SYSTEM VDMA_Station1_Emulator
  (* Version 1.0, 2021-08-05, dorofeev *)
  APPLICATION VDMA_Station1_EmulatorApp
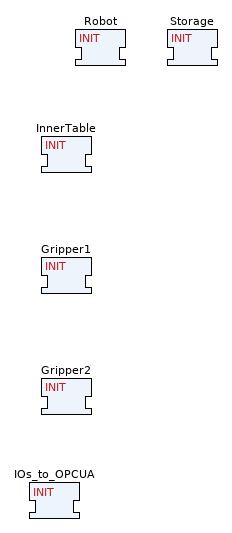
    SUBAPPLICATION Robot
      EVENT_INPUT
        INIT;
      END_EVENT
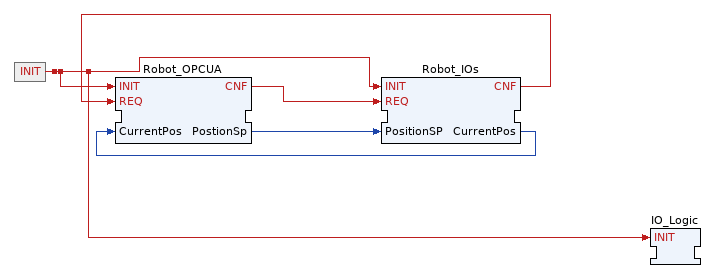
      SUBAPPLICATION IO_Logic
        EVENT_INPUT
          INIT;
        END_EVENT
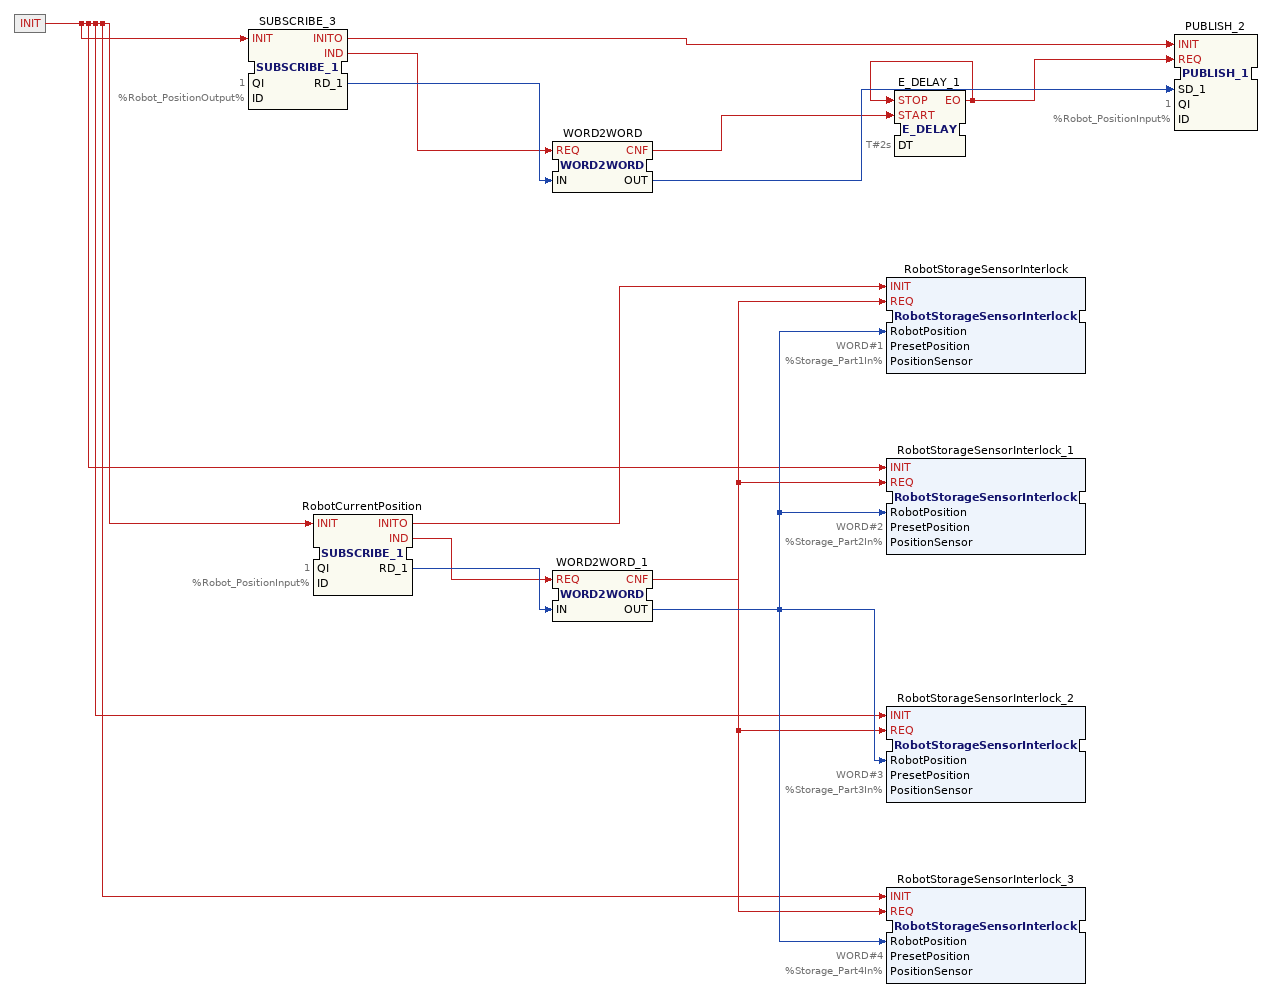
        FBS
          SUBSCRIBE_3 : SUBSCRIBE_1(QI := 1, ID := %Robot_PositionOutput%);
          E_DELAY_1 : E_DELAY(DT := T#2s);
          PUBLISH_2 : PUBLISH_1(QI := 1, ID := %Robot_PositionInput%);
          RobotCurrentPosition : SUBSCRIBE_1(QI := 1, ID := %Robot_PositionInput%);
          WORD2WORD_1 : WORD2WORD;
          WORD2WORD : WORD2WORD;
        END_FBS
        SUBAPPS
          RobotStorageSensorInterlock : RobotStorageSensorInterlock(PresetPosition := WORD#1, PositionSensor := %Storage_Part1In%);
          RobotStorageSensorInterlock_1 : RobotStorageSensorInterlock(PresetPosition := WORD#2, PositionSensor := %Storage_Part2In%);
          RobotStorageSensorInterlock_2 : RobotStorageSensorInterlock(PresetPosition := WORD#3, PositionSensor := %Storage_Part3In%);
          RobotStorageSensorInterlock_3 : RobotStorageSensorInterlock(PresetPosition := WORD#4, PositionSensor := %Storage_Part4In%);
        END_SUBAPPS
        EVENT_CONNECTIONS
          SUBSCRIBE_3.INITO TO PUBLISH_2.INIT;
          E_DELAY_1.EO TO E_DELAY_1.STOP;
          E_DELAY_1.EO TO PUBLISH_2.REQ;
          INIT TO SUBSCRIBE_3.INIT;
          INIT TO RobotStorageSensorInterlock_1.INIT;
          INIT TO RobotStorageSensorInterlock_2.INIT;
          INIT TO RobotStorageSensorInterlock_3.INIT;
          INIT TO RobotCurrentPosition.INIT;
          RobotCurrentPosition.INITO TO RobotStorageSensorInterlock.INIT;
          WORD2WORD_1.CNF TO RobotStorageSensorInterlock.REQ;
          WORD2WORD_1.CNF TO RobotStorageSensorInterlock_3.REQ;
          WORD2WORD_1.CNF TO RobotStorageSensorInterlock_2.REQ;
          WORD2WORD_1.CNF TO RobotStorageSensorInterlock_1.REQ;
          RobotCurrentPosition.IND TO WORD2WORD_1.REQ;
          SUBSCRIBE_3.IND TO WORD2WORD.REQ;
          WORD2WORD.CNF TO E_DELAY_1.START;
        END_CONNECTIONS
        DATA_CONNECTIONS
          WORD2WORD_1.OUT TO RobotStorageSensorInterlock_3.RobotPosition;
          WORD2WORD_1.OUT TO RobotStorageSensorInterlock_2.RobotPosition;
          WORD2WORD_1.OUT TO RobotStorageSensorInterlock_1.RobotPosition;
          WORD2WORD_1.OUT TO RobotStorageSensorInterlock.RobotPosition;
          RobotCurrentPosition.RD_1 TO WORD2WORD_1.IN;
          SUBSCRIBE_3.RD_1 TO WORD2WORD.IN;
          WORD2WORD.OUT TO PUBLISH_2.SD_1;
        END_CONNECTIONS
      END_SUBAPPLICATION
      SUBAPPLICATION Robot_OPCUA
        EVENT_INPUT
          INIT;
          REQ;
        END_EVENT
        EVENT_OUTPUT
          CNF;
        END_EVENT
        VAR_INPUT
          CurrentPos : WORD;
        END_VAR
        VAR_OUTPUT
          PostionSp : WORD;
        END_VAR
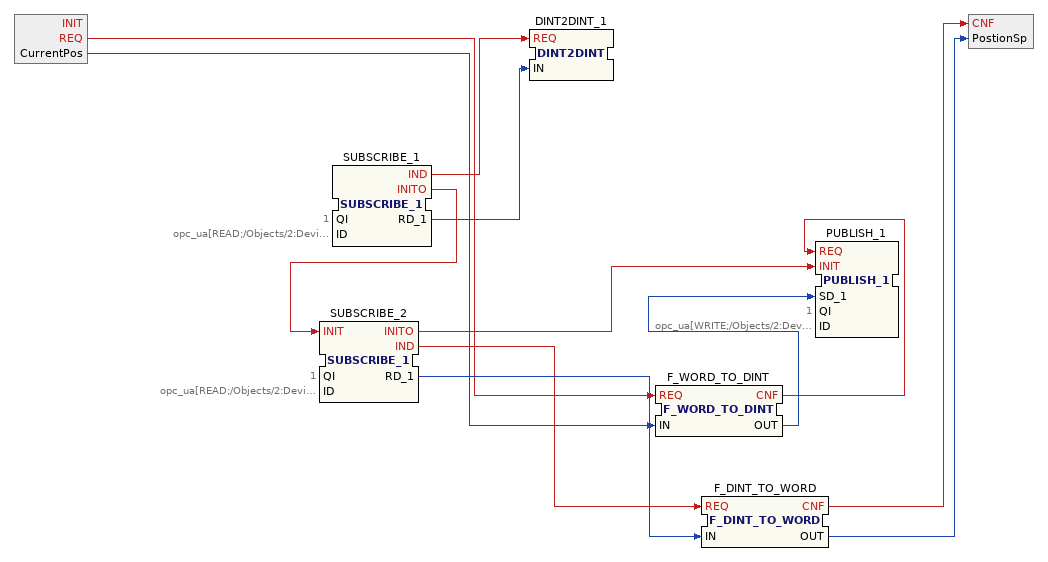
        FBS
          DINT2DINT_1 : DINT2DINT;
          F_WORD_TO_DINT : F_WORD_TO_DINT;
          SUBSCRIBE_2 : SUBSCRIBE_1(QI := 1, ID := opc_ua[READ;/Objects/2:DeviceSet/6:MotionDeviceSystem/5:ProcessData/6:VDMAINVARIABLES/6:SKILL_NMBR]);
          SUBSCRIBE_1 : SUBSCRIBE_1(QI := 1, ID := opc_ua[READ;/Objects/2:DeviceSet/6:MotionDeviceSystem/5:ProcessData/6:VDMAINVARIABLES/6:SKILL_CNTRL]);
          F_DINT_TO_WORD : F_DINT_TO_WORD;
          PUBLISH_1 : PUBLISH_1(QI := 1, ID := opc_ua[WRITE;/Objects/2:DeviceSet/6:MotionDeviceSystem/5:ProcessData/6:VDMAOUTVARIABLES/6:CURRENT_POSITION]);
        END_FBS
        EVENT_CONNECTIONS
          SUBSCRIBE_1.IND TO DINT2DINT_1.REQ;
          F_WORD_TO_DINT.CNF TO PUBLISH_1.REQ;
          SUBSCRIBE_1.INITO TO SUBSCRIBE_2.INIT;
          SUBSCRIBE_2.INITO TO PUBLISH_1.INIT;
          SUBSCRIBE_2.IND TO F_DINT_TO_WORD.REQ;
          REQ TO F_WORD_TO_DINT.REQ;
          F_DINT_TO_WORD.CNF TO CNF;
        END_CONNECTIONS
        DATA_CONNECTIONS
          SUBSCRIBE_1.RD_1 TO DINT2DINT_1.IN;
          F_WORD_TO_DINT.OUT TO PUBLISH_1.SD_1;
          SUBSCRIBE_2.RD_1 TO F_DINT_TO_WORD.IN;
          CurrentPos TO F_WORD_TO_DINT.IN;
          F_DINT_TO_WORD.OUT TO PostionSp;
        END_CONNECTIONS
      END_SUBAPPLICATION
      SUBAPPLICATION Robot_IOs
        EVENT_INPUT
          INIT;
          REQ;
        END_EVENT
        EVENT_OUTPUT
          CNF;
        END_EVENT
        VAR_INPUT
          PositionSP : WORD;
        END_VAR
        VAR_OUTPUT
          CurrentPos : WORD;
        END_VAR
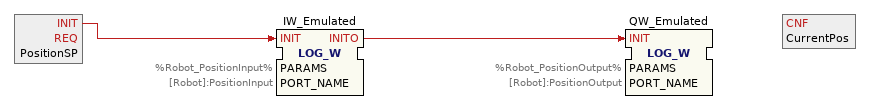
        FBS
          IW_Emulated : LOG_W(PARAMS := %Robot_PositionInput%, PORT_NAME := [Robot]:PositionInput);
          QW_Emulated : LOG_W(PARAMS := %Robot_PositionOutput%, PORT_NAME := [Robot]:PositionOutput);
        END_FBS
        EVENT_CONNECTIONS
          INIT TO IW_Emulated.INIT;
          IW_Emulated.INITO TO QW_Emulated.INIT;
        END_CONNECTIONS
      END_SUBAPPLICATION
      EVENT_CONNECTIONS
        INIT TO Robot_OPCUA.INIT;
        Robot_OPCUA.CNF TO Robot_IOs.REQ;
        INIT TO Robot_IOs.INIT;
        Robot_IOs.CNF TO Robot_OPCUA.REQ;
        INIT TO IO_Logic.INIT;
      END_CONNECTIONS
      DATA_CONNECTIONS
        Robot_OPCUA.PostionSp TO Robot_IOs.PositionSP;
        Robot_IOs.CurrentPos TO Robot_OPCUA.CurrentPos;
      END_CONNECTIONS
    END_SUBAPPLICATION
    SUBAPPLICATION InnerTable
      EVENT_INPUT
        INIT;
      END_EVENT
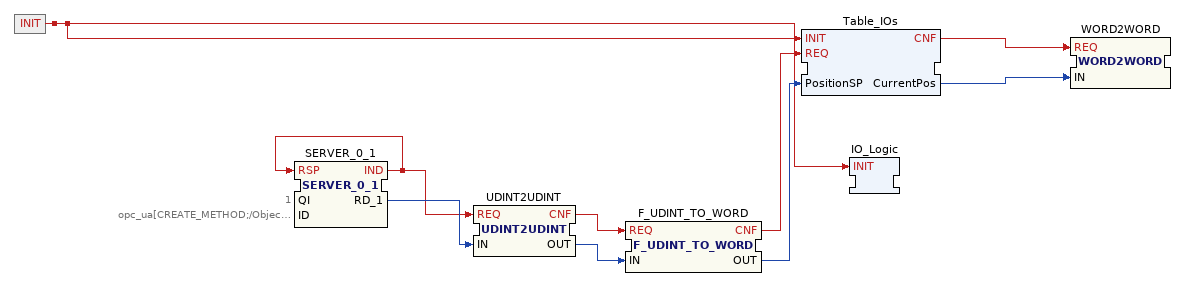
      FBS
        SERVER_0_1 : SERVER_0_1(QI := 1, ID := opc_ua[CREATE_METHOD;/Objects/7:WeissAxis/7:AxisSkillManager/7:MC_MovePresetPosition/7:SetStartParameter]);
        UDINT2UDINT : UDINT2UDINT;
        F_UDINT_TO_WORD : F_UDINT_TO_WORD;
        WORD2WORD : WORD2WORD;
      END_FBS
      SUBAPPLICATION IO_Logic
        EVENT_INPUT
          INIT;
        END_EVENT
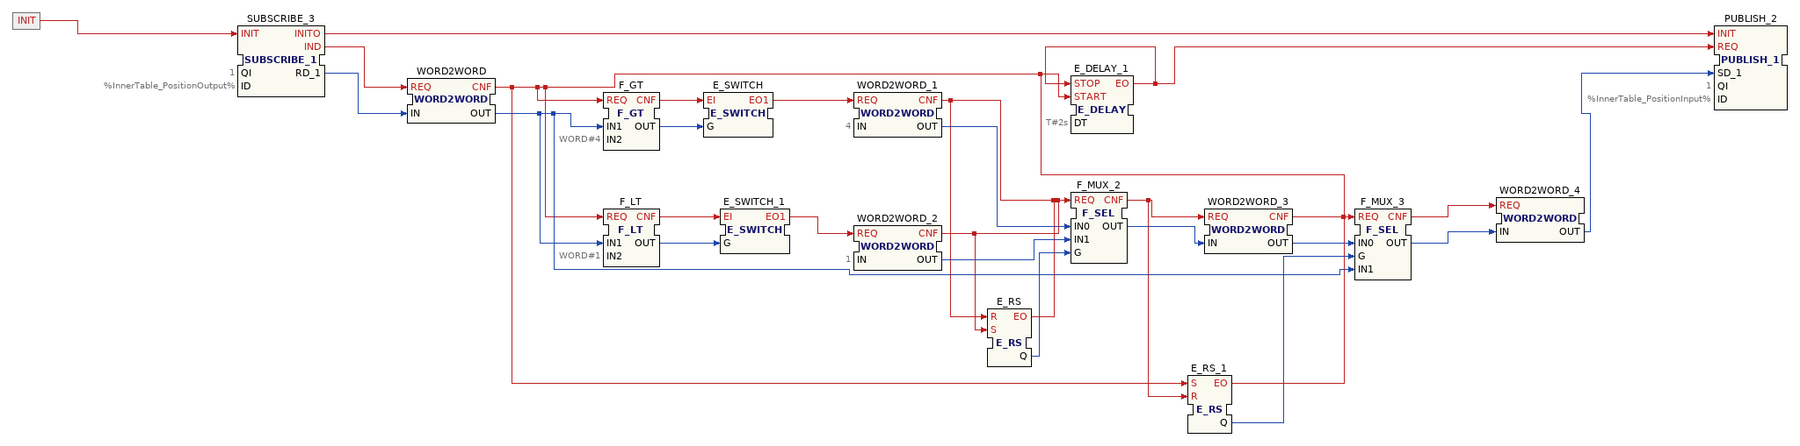
        FBS
          SUBSCRIBE_3 : SUBSCRIBE_1(QI := 1, ID := %InnerTable_PositionOutput%);
          WORD2WORD : WORD2WORD;
          E_DELAY_1 : E_DELAY(DT := T#2s);
          PUBLISH_2 : PUBLISH_1(QI := 1, ID := %InnerTable_PositionInput%);
          F_GT : F_GT(IN2 := WORD#4);
          F_LT : F_LT(IN2 := WORD#1);
          WORD2WORD_1 : WORD2WORD(IN := 4);
          WORD2WORD_2 : WORD2WORD(IN := 1);
          E_SWITCH : E_SWITCH;
          E_SWITCH_1 : E_SWITCH;
          WORD2WORD_3 : WORD2WORD;
          F_MUX_2 : F_SEL;
          F_MUX_3 : F_SEL;
          E_RS : E_RS;
          E_RS_1 : E_RS;
          WORD2WORD_4 : WORD2WORD;
        END_FBS
        EVENT_CONNECTIONS
          SUBSCRIBE_3.INITO TO PUBLISH_2.INIT;
          SUBSCRIBE_3.IND TO WORD2WORD.REQ;
          E_DELAY_1.EO TO E_DELAY_1.STOP;
          E_DELAY_1.EO TO PUBLISH_2.REQ;
          INIT TO SUBSCRIBE_3.INIT;
          WORD2WORD.CNF TO F_GT.REQ;
          WORD2WORD.CNF TO F_LT.REQ;
          F_GT.CNF TO E_SWITCH.EI;
          E_SWITCH.EO1 TO WORD2WORD_1.REQ;
          F_LT.CNF TO E_SWITCH_1.EI;
          E_SWITCH_1.EO1 TO WORD2WORD_2.REQ;
          WORD2WORD.CNF TO E_DELAY_1.START;
          WORD2WORD_1.CNF TO F_MUX_2.REQ;
          WORD2WORD_2.CNF TO F_MUX_2.REQ;
          F_MUX_2.CNF TO WORD2WORD_3.REQ;
          WORD2WORD_3.CNF TO F_MUX_3.REQ;
          WORD2WORD_1.CNF TO E_RS.R;
          WORD2WORD_2.CNF TO E_RS.S;
          E_RS.EO TO F_MUX_2.REQ;
          WORD2WORD.CNF TO E_RS_1.S;
          F_MUX_2.CNF TO E_RS_1.R;
          E_RS_1.EO TO F_MUX_3.REQ;
          F_MUX_3.CNF TO WORD2WORD_4.REQ;
          WORD2WORD.CNF TO F_MUX_3.REQ;
        END_CONNECTIONS
        DATA_CONNECTIONS
          SUBSCRIBE_3.RD_1 TO WORD2WORD.IN;
          WORD2WORD.OUT TO F_LT.IN1;
          WORD2WORD.OUT TO F_GT.IN1;
          F_GT.OUT TO E_SWITCH.G;
          F_LT.OUT TO E_SWITCH_1.G;
          F_MUX_2.OUT TO WORD2WORD_3.IN;
          WORD2WORD_1.OUT TO F_MUX_2.IN0;
          WORD2WORD_2.OUT TO F_MUX_2.IN1;
          WORD2WORD_3.OUT TO F_MUX_3.IN0;
          E_RS.Q TO F_MUX_2.G;
          E_RS_1.Q TO F_MUX_3.G;
          WORD2WORD.OUT TO F_MUX_3.IN1;
          F_MUX_3.OUT TO WORD2WORD_4.IN;
          WORD2WORD_4.OUT TO PUBLISH_2.SD_1;
        END_CONNECTIONS
      END_SUBAPPLICATION
      SUBAPPLICATION Table_IOs
        EVENT_INPUT
          INIT;
          REQ;
        END_EVENT
        EVENT_OUTPUT
          CNF;
        END_EVENT
        VAR_INPUT
          PositionSP : WORD;
        END_VAR
        VAR_OUTPUT
          CurrentPos : WORD;
        END_VAR
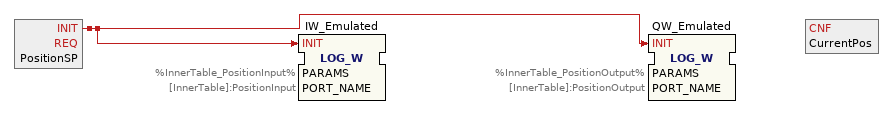
        FBS
          IW_Emulated : LOG_W(PARAMS := %InnerTable_PositionInput%, PORT_NAME := [InnerTable]:PositionInput);
          QW_Emulated : LOG_W(PARAMS := %InnerTable_PositionOutput%, PORT_NAME := [InnerTable]:PositionOutput);
        END_FBS
        EVENT_CONNECTIONS
          INIT TO IW_Emulated.INIT;
          INIT TO QW_Emulated.INIT;
        END_CONNECTIONS
      END_SUBAPPLICATION
      EVENT_CONNECTIONS
        SERVER_0_1.IND TO UDINT2UDINT.REQ;
        INIT TO Table_IOs.INIT;
        INIT TO IO_Logic.INIT;
        UDINT2UDINT.CNF TO F_UDINT_TO_WORD.REQ;
        F_UDINT_TO_WORD.CNF TO Table_IOs.REQ;
        Table_IOs.CNF TO WORD2WORD.REQ;
        SERVER_0_1.IND TO SERVER_0_1.RSP;
      END_CONNECTIONS
      DATA_CONNECTIONS
        SERVER_0_1.RD_1 TO UDINT2UDINT.IN;
        UDINT2UDINT.OUT TO F_UDINT_TO_WORD.IN;
        F_UDINT_TO_WORD.OUT TO Table_IOs.PositionSP;
        Table_IOs.CurrentPos TO WORD2WORD.IN;
      END_CONNECTIONS
    END_SUBAPPLICATION
    SUBAPPLICATION Storage
      EVENT_INPUT
        INIT;
      END_EVENT
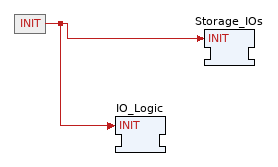
      SUBAPPLICATION IO_Logic
        EVENT_INPUT
          INIT;
        END_EVENT
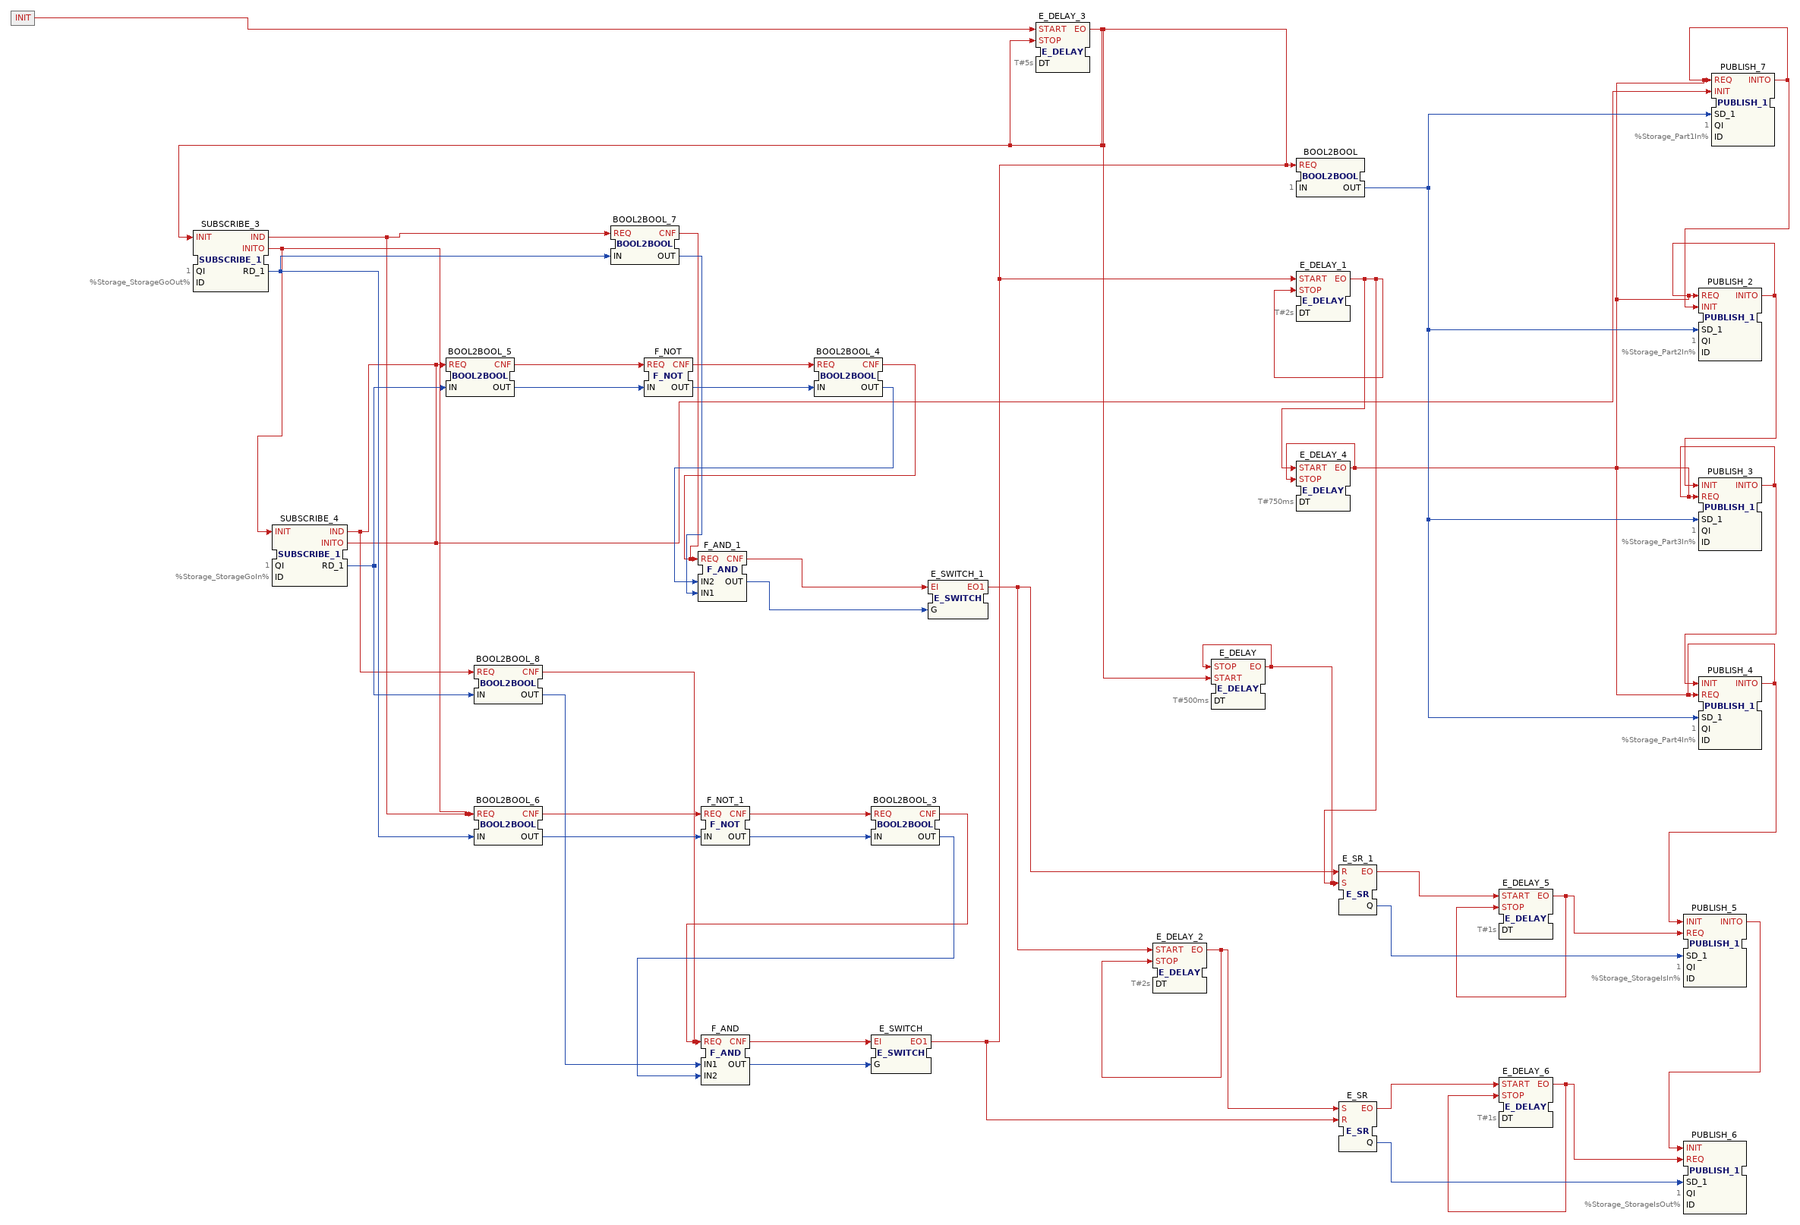
        FBS
          E_SWITCH_1 : E_SWITCH;
          BOOL2BOOL_4 : BOOL2BOOL;
          F_NOT : F_NOT;
          PUBLISH_3 : PUBLISH_1(QI := 1, ID := %Storage_Part3In%);
          BOOL2BOOL_6 : BOOL2BOOL;
          E_SR_1 : E_SR;
          F_NOT_1 : F_NOT;
          PUBLISH_7 : PUBLISH_1(QI := 1, ID := %Storage_Part1In%);
          BOOL2BOOL : BOOL2BOOL(IN := 1);
          BOOL2BOOL_5 : BOOL2BOOL;
          BOOL2BOOL_7 : BOOL2BOOL;
          E_SR : E_SR;
          F_AND_1 : F_AND;
          SUBSCRIBE_4 : SUBSCRIBE_1(QI := 1, ID := %Storage_StorageGoIn%);
          SUBSCRIBE_3 : SUBSCRIBE_1(QI := 1, ID := %Storage_StorageGoOut%);
          PUBLISH_6 : PUBLISH_1(QI := 1, ID := %Storage_StorageIsOut%);
          F_AND : F_AND;
          BOOL2BOOL_3 : BOOL2BOOL;
          PUBLISH_5 : PUBLISH_1(QI := 1, ID := %Storage_StorageIsIn%);
          PUBLISH_4 : PUBLISH_1(QI := 1, ID := %Storage_Part4In%);
          E_DELAY_2 : E_DELAY(DT := T#2s);
          BOOL2BOOL_8 : BOOL2BOOL;
          E_DELAY_1 : E_DELAY(DT := T#2s);
          PUBLISH_2 : PUBLISH_1(QI := 1, ID := %Storage_Part2In%);
          E_SWITCH : E_SWITCH;
          E_DELAY : E_DELAY(DT := T#500ms);
          E_DELAY_3 : E_DELAY(DT := T#5s);
          E_DELAY_4 : E_DELAY(DT := T#750ms);
          E_DELAY_5 : E_DELAY(DT := T#1s);
          E_DELAY_6 : E_DELAY(DT := T#1s);
        END_FBS
        EVENT_CONNECTIONS
          F_AND_1.CNF TO E_SWITCH_1.EI;
          E_SWITCH_1.EO1 TO E_SR_1.R;
          E_SWITCH_1.EO1 TO E_DELAY_2.START;
          F_NOT.CNF TO BOOL2BOOL_4.REQ;
          BOOL2BOOL_4.CNF TO F_AND_1.REQ;
          BOOL2BOOL_5.CNF TO F_NOT.REQ;
          PUBLISH_2.INITO TO PUBLISH_3.INIT;
          PUBLISH_3.INITO TO PUBLISH_3.REQ;
          PUBLISH_3.INITO TO PUBLISH_4.INIT;
          SUBSCRIBE_3.IND TO BOOL2BOOL_6.REQ;
          SUBSCRIBE_3.INITO TO BOOL2BOOL_6.REQ;
          BOOL2BOOL_6.CNF TO F_NOT_1.REQ;
          E_DELAY_1.EO TO E_SR_1.S;
          F_NOT_1.CNF TO BOOL2BOOL_3.REQ;
          PUBLISH_7.INITO TO PUBLISH_7.REQ;
          E_SWITCH.EO1 TO BOOL2BOOL.REQ;
          SUBSCRIBE_4.IND TO BOOL2BOOL_5.REQ;
          SUBSCRIBE_4.INITO TO BOOL2BOOL_5.REQ;
          SUBSCRIBE_3.IND TO BOOL2BOOL_7.REQ;
          BOOL2BOOL_7.CNF TO F_AND_1.REQ;
          E_DELAY_2.EO TO E_SR.S;
          E_SWITCH.EO1 TO E_SR.R;
          SUBSCRIBE_3.INITO TO SUBSCRIBE_4.INIT;
          SUBSCRIBE_4.IND TO BOOL2BOOL_8.REQ;
          PUBLISH_5.INITO TO PUBLISH_6.INIT;
          BOOL2BOOL_3.CNF TO F_AND.REQ;
          BOOL2BOOL_8.CNF TO F_AND.REQ;
          F_AND.CNF TO E_SWITCH.EI;
          PUBLISH_4.INITO TO PUBLISH_5.INIT;
          PUBLISH_4.INITO TO PUBLISH_4.REQ;
          E_DELAY_2.EO TO E_DELAY_2.STOP;
          E_SWITCH.EO1 TO E_DELAY_1.START;
          E_DELAY_1.EO TO E_DELAY_1.STOP;
          PUBLISH_2.INITO TO PUBLISH_2.REQ;
          E_DELAY.EO TO E_DELAY.STOP;
          E_DELAY.EO TO E_SR_1.S;
          E_DELAY_3.EO TO BOOL2BOOL.REQ;
          E_DELAY_3.EO TO E_DELAY.START;
          INIT TO E_DELAY_3.START;
          E_DELAY_3.EO TO E_DELAY_3.STOP;
          E_DELAY_4.EO TO PUBLISH_2.REQ;
          E_DELAY_4.EO TO PUBLISH_4.REQ;
          E_DELAY_4.EO TO PUBLISH_7.REQ;
          E_DELAY_4.EO TO PUBLISH_3.REQ;
          E_DELAY_1.EO TO E_DELAY_4.START;
          E_DELAY_4.EO TO E_DELAY_4.STOP;
          E_SR_1.EO TO E_DELAY_5.START;
          E_DELAY_5.EO TO PUBLISH_5.REQ;
          E_DELAY_5.EO TO E_DELAY_5.STOP;
          E_SR.EO TO E_DELAY_6.START;
          E_DELAY_6.EO TO PUBLISH_6.REQ;
          E_DELAY_6.EO TO E_DELAY_6.STOP;
          E_DELAY_3.EO TO SUBSCRIBE_3.INIT;
          PUBLISH_7.INITO TO PUBLISH_2.INIT;
          SUBSCRIBE_4.INITO TO PUBLISH_7.INIT;
        END_CONNECTIONS
        DATA_CONNECTIONS
          F_AND_1.OUT TO E_SWITCH_1.G;
          F_NOT.OUT TO BOOL2BOOL_4.IN;
          BOOL2BOOL_4.OUT TO F_AND_1.IN2;
          BOOL2BOOL_5.OUT TO F_NOT.IN;
          BOOL2BOOL.OUT TO PUBLISH_3.SD_1;
          SUBSCRIBE_3.RD_1 TO BOOL2BOOL_6.IN;
          BOOL2BOOL_6.OUT TO F_NOT_1.IN;
          F_NOT_1.OUT TO BOOL2BOOL_3.IN;
          BOOL2BOOL.OUT TO PUBLISH_7.SD_1;
          BOOL2BOOL.OUT TO PUBLISH_4.SD_1;
          BOOL2BOOL.OUT TO PUBLISH_2.SD_1;
          SUBSCRIBE_4.RD_1 TO BOOL2BOOL_5.IN;
          SUBSCRIBE_3.RD_1 TO BOOL2BOOL_7.IN;
          BOOL2BOOL_7.OUT TO F_AND_1.IN1;
          E_SR.Q TO PUBLISH_6.SD_1;
          SUBSCRIBE_4.RD_1 TO BOOL2BOOL_8.IN;
          BOOL2BOOL_8.OUT TO F_AND.IN1;
          BOOL2BOOL_3.OUT TO F_AND.IN2;
          F_AND.OUT TO E_SWITCH.G;
          E_SR_1.Q TO PUBLISH_5.SD_1;
        END_CONNECTIONS
      END_SUBAPPLICATION
      SUBAPPLICATION Storage_IOs
        EVENT_INPUT
          INIT;
        END_EVENT
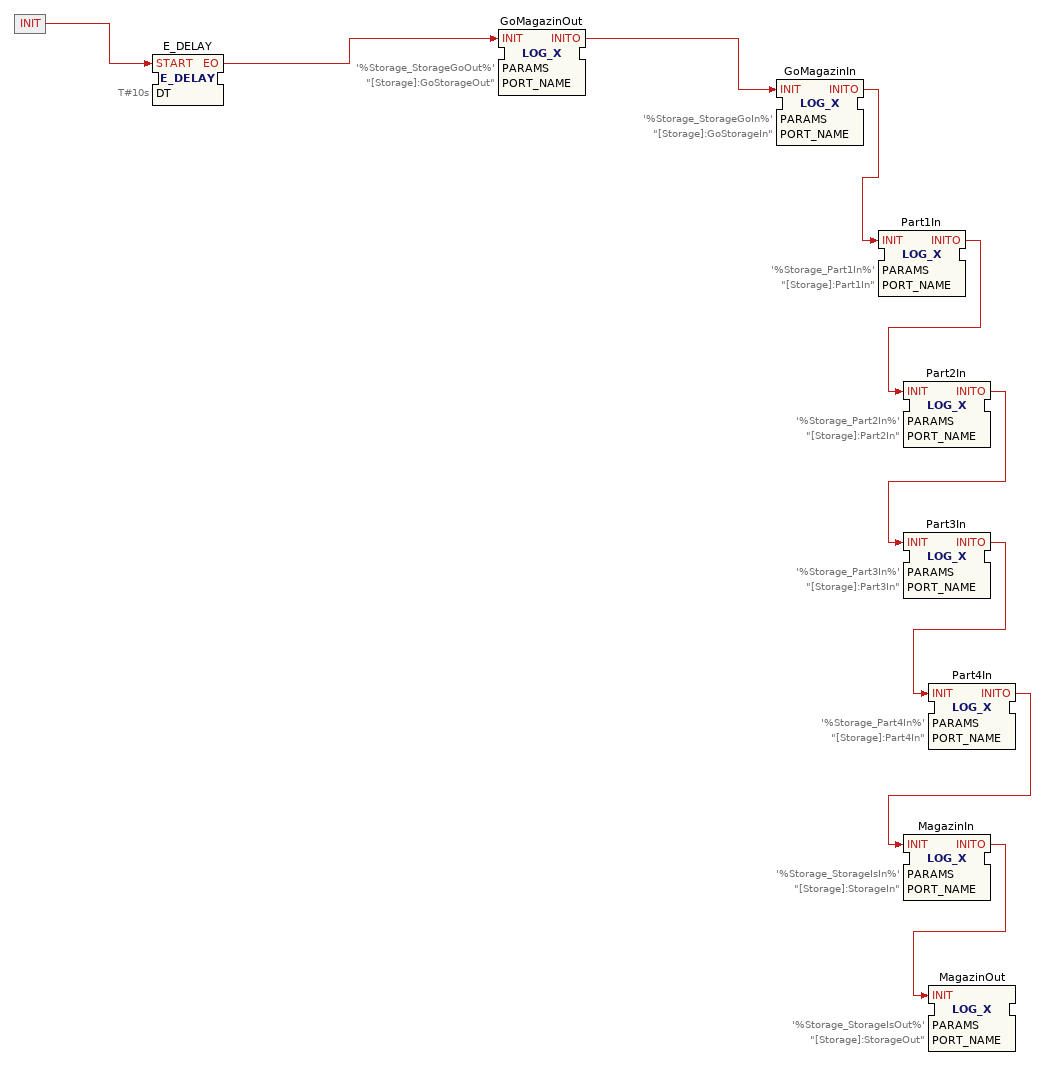
        FBS
          GoMagazinIn : LOG_X(PARAMS := '%Storage_StorageGoIn%', PORT_NAME := "[Storage]:GoStorageIn");
          GoMagazinOut : LOG_X(PARAMS := '%Storage_StorageGoOut%', PORT_NAME := "[Storage]:GoStorageOut");
          Part2In : LOG_X(PARAMS := '%Storage_Part2In%', PORT_NAME := "[Storage]:Part2In");
          Part1In : LOG_X(PARAMS := '%Storage_Part1In%', PORT_NAME := "[Storage]:Part1In");
          Part4In : LOG_X(PARAMS := '%Storage_Part4In%', PORT_NAME := "[Storage]:Part4In");
          Part3In : LOG_X(PARAMS := '%Storage_Part3In%', PORT_NAME := "[Storage]:Part3In");
          MagazinIn : LOG_X(PARAMS := '%Storage_StorageIsIn%', PORT_NAME := "[Storage]:StorageIn");
          MagazinOut : LOG_X(PARAMS := '%Storage_StorageIsOut%', PORT_NAME := "[Storage]:StorageOut");
          E_DELAY : E_DELAY(DT := T#10s);
        END_FBS
        EVENT_CONNECTIONS
          GoMagazinOut.INITO TO GoMagazinIn.INIT;
          GoMagazinIn.INITO TO Part1In.INIT;
          Part1In.INITO TO Part2In.INIT;
          Part2In.INITO TO Part3In.INIT;
          Part3In.INITO TO Part4In.INIT;
          Part4In.INITO TO MagazinIn.INIT;
          MagazinIn.INITO TO MagazinOut.INIT;
          INIT TO E_DELAY.START;
          E_DELAY.EO TO GoMagazinOut.INIT;
        END_CONNECTIONS
      END_SUBAPPLICATION
      EVENT_CONNECTIONS
        INIT TO IO_Logic.INIT;
        INIT TO Storage_IOs.INIT;
      END_CONNECTIONS
    END_SUBAPPLICATION
    SUBAPPLICATION Gripper1
      EVENT_INPUT
        INIT;
      END_EVENT
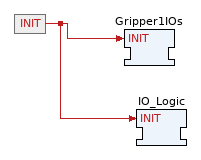
      SUBAPPLICATION Gripper1IOs
        EVENT_INPUT
          INIT;
        END_EVENT
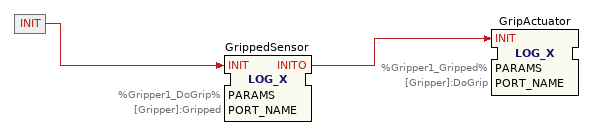
        FBS
          GripActuator : LOG_X(PARAMS := %Gripper1_Gripped%, PORT_NAME := [Gripper]:DoGrip);
          GrippedSensor : LOG_X(PARAMS := %Gripper1_DoGrip%, PORT_NAME := [Gripper]:Gripped);
        END_FBS
        EVENT_CONNECTIONS
          INIT TO GrippedSensor.INIT;
          GrippedSensor.INITO TO GripActuator.INIT;
        END_CONNECTIONS
      END_SUBAPPLICATION
      SUBAPPLICATION IO_Logic
        EVENT_INPUT
          INIT;
        END_EVENT
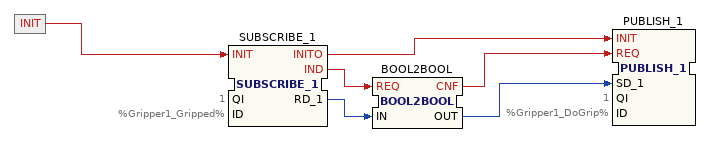
        FBS
          SUBSCRIBE_1 : SUBSCRIBE_1(QI := 1, ID := %Gripper1_Gripped%);
          BOOL2BOOL : BOOL2BOOL;
          PUBLISH_1 : PUBLISH_1(QI := 1, ID := %Gripper1_DoGrip%);
        END_FBS
        EVENT_CONNECTIONS
          SUBSCRIBE_1.INITO TO PUBLISH_1.INIT;
          SUBSCRIBE_1.IND TO BOOL2BOOL.REQ;
          BOOL2BOOL.CNF TO PUBLISH_1.REQ;
          INIT TO SUBSCRIBE_1.INIT;
        END_CONNECTIONS
        DATA_CONNECTIONS
          SUBSCRIBE_1.RD_1 TO BOOL2BOOL.IN;
          BOOL2BOOL.OUT TO PUBLISH_1.SD_1;
        END_CONNECTIONS
      END_SUBAPPLICATION
      EVENT_CONNECTIONS
        INIT TO IO_Logic.INIT;
        INIT TO Gripper1IOs.INIT;
      END_CONNECTIONS
    END_SUBAPPLICATION
    SUBAPPLICATION Gripper2
      EVENT_INPUT
        INIT;
      END_EVENT
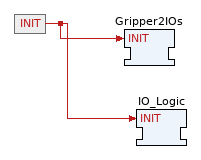
      SUBAPPLICATION Gripper2IOs
        EVENT_INPUT
          INIT;
        END_EVENT
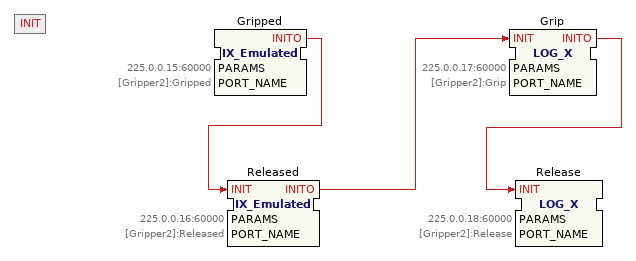
        FBS
          Grip : LOG_X(PARAMS := 225.0.0.17:60000, PORT_NAME := [Gripper2]:Grip);
          Gripped : IX_Emulated(PARAMS := 225.0.0.15:60000, PORT_NAME := [Gripper2]:Gripped);
          Released : IX_Emulated(PARAMS := 225.0.0.16:60000, PORT_NAME := [Gripper2]:Released);
          Release : LOG_X(PARAMS := 225.0.0.18:60000, PORT_NAME := [Gripper2]:Release);
        END_FBS
        EVENT_CONNECTIONS
          Gripped.INITO TO Released.INIT;
          Released.INITO TO Grip.INIT;
          Grip.INITO TO Release.INIT;
        END_CONNECTIONS
      END_SUBAPPLICATION
      SUBAPPLICATION IO_Logic
        EVENT_INPUT
          INIT;
        END_EVENT
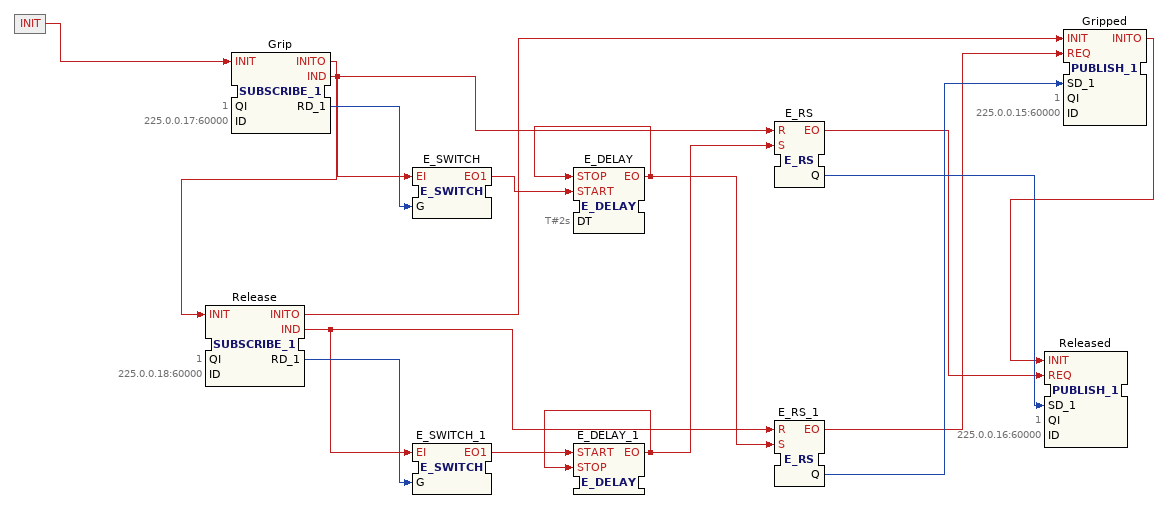
        FBS
          Grip : SUBSCRIBE_1(QI := 1, ID := 225.0.0.17:60000);
          Gripped : PUBLISH_1(QI := 1, ID := 225.0.0.15:60000);
          Release : SUBSCRIBE_1(QI := 1, ID := 225.0.0.18:60000);
          Released : PUBLISH_1(QI := 1, ID := 225.0.0.16:60000);
          E_DELAY : E_DELAY(DT := T#2s);
          E_RS : E_RS;
          E_RS_1 : E_RS;
          E_DELAY_1 : E_DELAY;
          E_SWITCH : E_SWITCH;
          E_SWITCH_1 : E_SWITCH;
        END_FBS
        EVENT_CONNECTIONS
          INIT TO Grip.INIT;
          Grip.INITO TO Release.INIT;
          Release.INITO TO Gripped.INIT;
          Gripped.INITO TO Released.INIT;
          E_DELAY.EO TO E_DELAY.STOP;
          Grip.IND TO E_RS.R;
          E_RS.EO TO Released.REQ;
          Release.IND TO E_RS_1.R;
          E_RS_1.EO TO Gripped.REQ;
          E_DELAY.EO TO E_RS_1.S;
          Grip.IND TO E_SWITCH.EI;
          E_SWITCH.EO1 TO E_DELAY.START;
          Release.IND TO E_SWITCH_1.EI;
          E_SWITCH_1.EO1 TO E_DELAY_1.START;
          E_DELAY_1.EO TO E_DELAY_1.STOP;
          E_DELAY_1.EO TO E_RS.S;
        END_CONNECTIONS
        DATA_CONNECTIONS
          E_RS.Q TO Released.SD_1;
          E_RS_1.Q TO Gripped.SD_1;
          Grip.RD_1 TO E_SWITCH.G;
          Release.RD_1 TO E_SWITCH_1.G;
        END_CONNECTIONS
      END_SUBAPPLICATION
      EVENT_CONNECTIONS
        INIT TO Gripper2IOs.INIT;
        INIT TO IO_Logic.INIT;
      END_CONNECTIONS
    END_SUBAPPLICATION
    SUBAPPLICATION IOs_to_OPCUA
      EVENT_INPUT
        INIT;
      END_EVENT
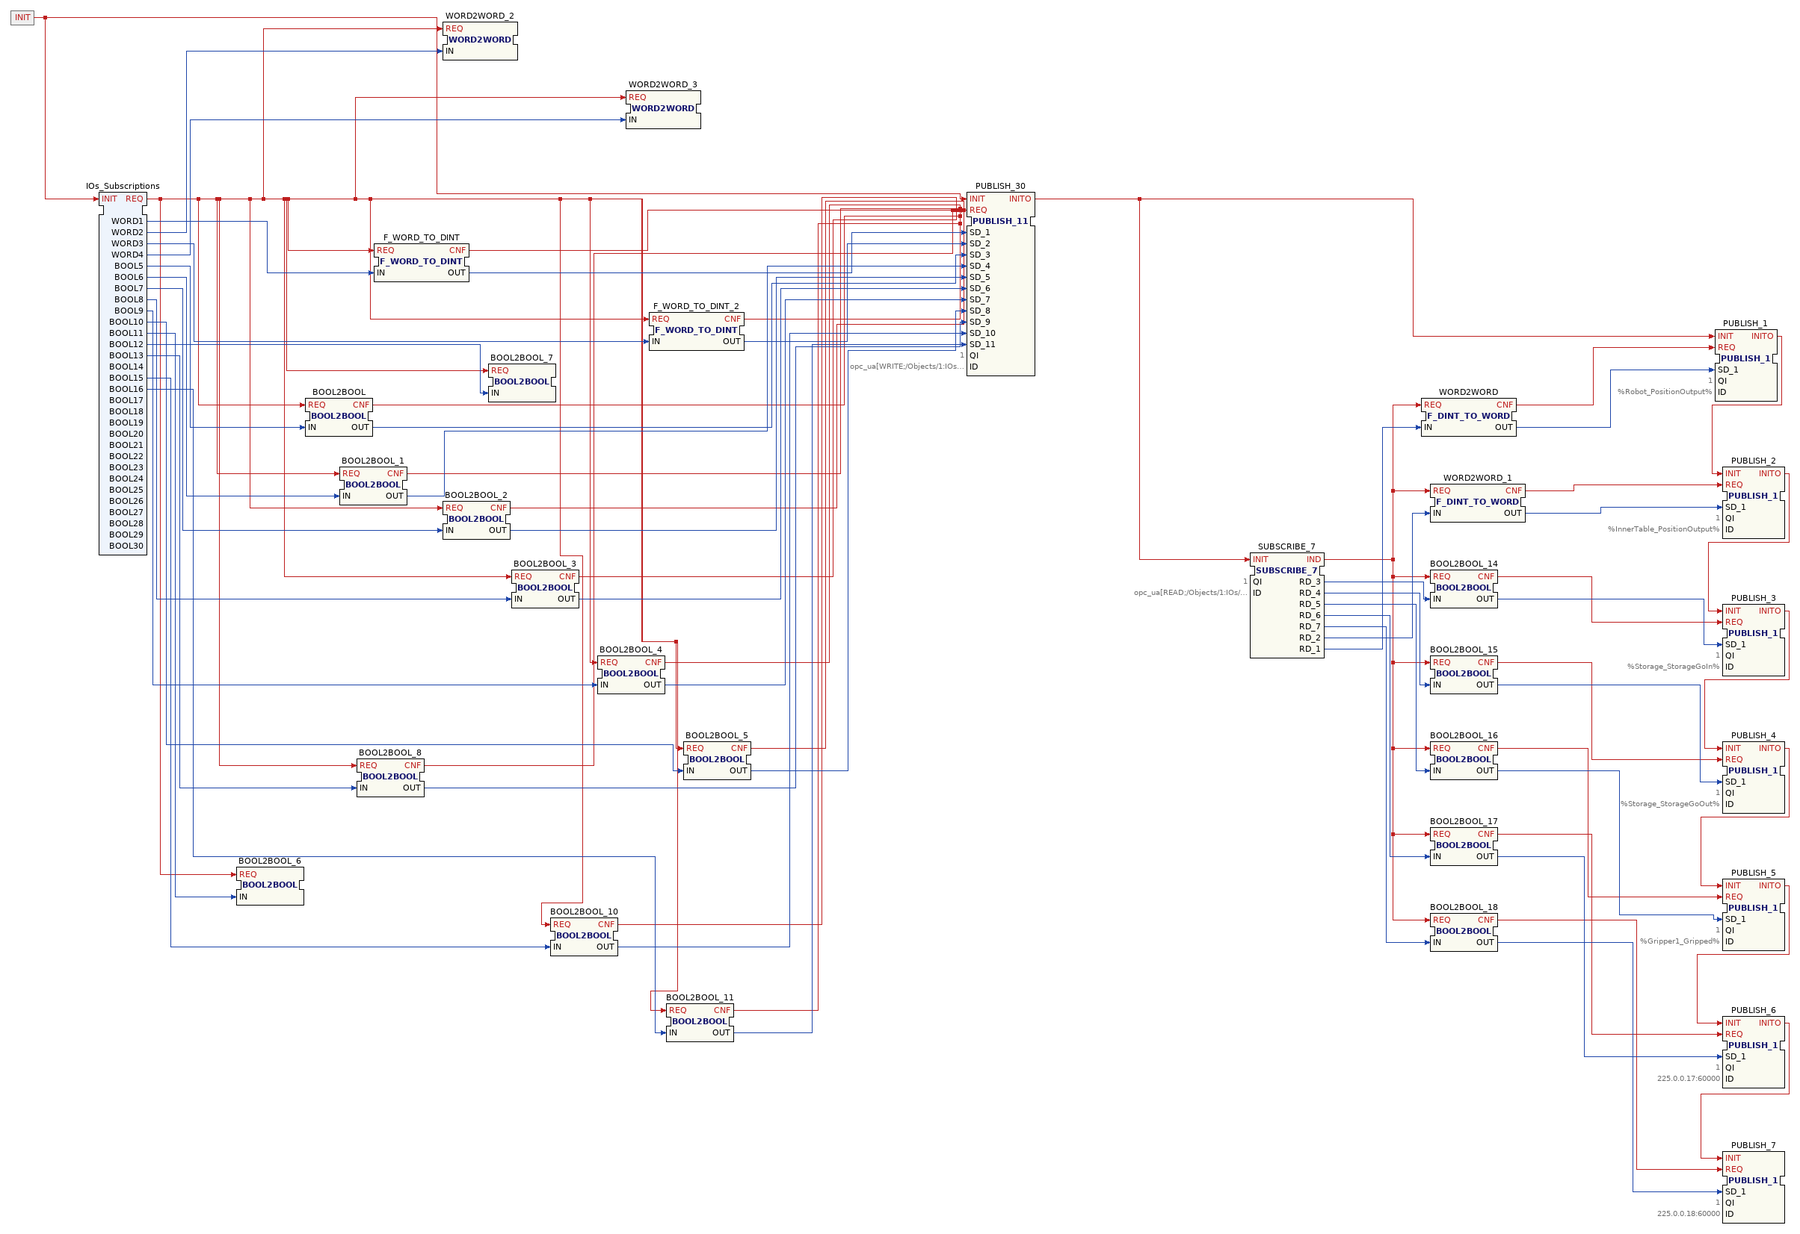
      FBS
        F_WORD_TO_DINT : F_WORD_TO_DINT;
        F_WORD_TO_DINT_2 : F_WORD_TO_DINT;
        BOOL2BOOL : BOOL2BOOL;
        BOOL2BOOL_1 : BOOL2BOOL;
        BOOL2BOOL_2 : BOOL2BOOL;
        BOOL2BOOL_3 : BOOL2BOOL;
        BOOL2BOOL_4 : BOOL2BOOL;
        BOOL2BOOL_5 : BOOL2BOOL;
        BOOL2BOOL_8 : BOOL2BOOL;
        BOOL2BOOL_10 : BOOL2BOOL;
        BOOL2BOOL_11 : BOOL2BOOL;
        SUBSCRIBE_7 : SUBSCRIBE_7(QI := 1, ID := opc_ua[READ;/Objects/1:IOs/1:Robot.PresetPosition;/Objects/1:IOs/1:InnerTable.PresetPosition;/Objects/1:IOs/1:Storage.GoMagazinIn;/Objects/1:IOs/1:Storage.GoMagazinOut;/Objects/1:IOs/1:Gripper1.Grip;/Objects/1:IOs/1:Gripper2.Grip;/Objects/1:IOs/1:Gripper2.Release]);
        BOOL2BOOL_14 : BOOL2BOOL;
        BOOL2BOOL_15 : BOOL2BOOL;
        BOOL2BOOL_16 : BOOL2BOOL;
        BOOL2BOOL_17 : BOOL2BOOL;
        BOOL2BOOL_18 : BOOL2BOOL;
        PUBLISH_1 : PUBLISH_1(QI := 1, ID := %Robot_PositionOutput%);
        PUBLISH_2 : PUBLISH_1(QI := 1, ID := %InnerTable_PositionOutput%);
        PUBLISH_3 : PUBLISH_1(QI := 1, ID := %Storage_StorageGoIn%);
        PUBLISH_4 : PUBLISH_1(QI := 1, ID := %Storage_StorageGoOut%);
        PUBLISH_5 : PUBLISH_1(QI := 1, ID := %Gripper1_Gripped%);
        PUBLISH_6 : PUBLISH_1(QI := 1, ID := 225.0.0.17:60000);
        PUBLISH_7 : PUBLISH_1(QI := 1, ID := 225.0.0.18:60000);
        PUBLISH_30 : PUBLISH_11(QI := 1, ID := opc_ua[WRITE;/Objects/1:IOs/1:Robot.CurrentPosition;/Objects/1:IOs/1:InnerTable.CurrentPosition;/Objects/1:IOs/1:Storage.Part1In;/Objects/1:IOs/1:Storage.Part2In;/Objects/1:IOs/1:Storage.Part3In;/Objects/1:IOs/1:Storage.Part4In;/Objects/1:IOs/1:Storage.MagazinIn;/Objects/1:IOs/1:Storage.MagazinOut;/Objects/1:IOs/1:Gripper1.Gripped;/Objects/1:IOs/1:Gripper2.Gripped;/Objects/1:IOs/1:Gripper2.Released]);
        WORD2WORD_1 : F_DINT_TO_WORD;
        WORD2WORD : F_DINT_TO_WORD;
        WORD2WORD_2 : WORD2WORD;
        WORD2WORD_3 : WORD2WORD;
        BOOL2BOOL_6 : BOOL2BOOL;
        BOOL2BOOL_7 : BOOL2BOOL;
      END_FBS
      SUBAPPLICATION IOs_Subscriptions
        EVENT_INPUT
          INIT;
        END_EVENT
        EVENT_OUTPUT
          REQ;
        END_EVENT
        VAR_OUTPUT
          WORD1 : WORD;
          WORD2 : WORD;
          WORD3 : WORD;
          WORD4 : WORD;
          BOOL5 : BOOL;
          BOOL6 : BOOL;
          BOOL7 : BOOL;
          BOOL8 : BOOL;
          BOOL9 : BOOL;
          BOOL10 : BOOL;
          BOOL11 : BOOL;
          BOOL12 : BOOL;
          BOOL13 : BOOL;
          BOOL14 : BOOL;
          BOOL15 : BOOL;
          BOOL16 : BOOL;
          BOOL17 : BOOL;
          BOOL18 : BOOL;
          BOOL19 : BOOL;
          BOOL20 : BOOL;
          BOOL21 : BOOL;
          BOOL22 : BOOL;
          BOOL23 : BOOL;
          BOOL24 : BOOL;
          BOOL25 : BOOL;
          BOOL26 : BOOL;
          BOOL27 : BOOL;
          BOOL28 : BOOL;
          BOOL29 : BOOL;
          BOOL30 : BOOL;
        END_VAR
        FBS
          SUBSCRIBE_1 : SUBSCRIBE_1(QI := 1, ID := %Robot_PositionInput%);
          SUBSCRIBE_2 : SUBSCRIBE_1(QI := 1, ID := %Robot_PositionOutput%);
          SUBSCRIBE_3 : SUBSCRIBE_1(QI := 1, ID := %InnerTable_PositionInput%);
          SUBSCRIBE_4 : SUBSCRIBE_1(QI := 1, ID := %InnerTable_PositionOutput%);
          SUBSCRIBE_5 : SUBSCRIBE_1(QI := 1, ID := %Storage_Part1In%);
          SUBSCRIBE_6 : SUBSCRIBE_1(QI := 1, ID := %Storage_Part2In%);
          SUBSCRIBE_7 : SUBSCRIBE_1(QI := 1, ID := %Storage_Part3In%);
          SUBSCRIBE_8 : SUBSCRIBE_1(QI := 1, ID := %Storage_Part4In%);
          SUBSCRIBE_9 : SUBSCRIBE_1(QI := 1, ID := %Storage_StorageIsIn%);
          SUBSCRIBE_10 : SUBSCRIBE_1(QI := 1, ID := %Storage_StorageIsOut%);
          SUBSCRIBE_11 : SUBSCRIBE_1(QI := 1, ID := %Storage_StorageGoOut%);
          SUBSCRIBE_12 : SUBSCRIBE_1(QI := 1, ID := %Storage_StorageGoIn%);
          SUBSCRIBE_13 : SUBSCRIBE_1(QI := 1, ID := %Gripper1_DoGrip%);
          SUBSCRIBE_14 : SUBSCRIBE_1(QI := 1, ID := %Gripper1_Gripped%);
          SUBSCRIBE_15 : SUBSCRIBE_1(QI := 1, ID := 225.0.0.15:60000);
          SUBSCRIBE_16 : SUBSCRIBE_1(QI := 1, ID := 225.0.0.16:60000);
          SUBSCRIBE_17 : SUBSCRIBE_1(QI := 1, ID := 225.0.0.17:60000);
          SUBSCRIBE_18 : SUBSCRIBE_1(QI := 1, ID := 225.0.0.18:60000);
          SUBSCRIBE_19 : SUBSCRIBE_1;
          SUBSCRIBE_20 : SUBSCRIBE_1;
          SUBSCRIBE_21 : SUBSCRIBE_1;
          SUBSCRIBE_22 : SUBSCRIBE_1;
          SUBSCRIBE_23 : SUBSCRIBE_1;
          SUBSCRIBE_24 : SUBSCRIBE_1;
          SUBSCRIBE_25 : SUBSCRIBE_1;
          SUBSCRIBE_26 : SUBSCRIBE_1;
          SUBSCRIBE_27 : SUBSCRIBE_1;
          SUBSCRIBE_28 : SUBSCRIBE_1;
          SUBSCRIBE_29 : SUBSCRIBE_1;
          SUBSCRIBE_30 : SUBSCRIBE_1;
        END_FBS
        EVENT_CONNECTIONS
          SUBSCRIBE_1.IND TO REQ;
          SUBSCRIBE_2.IND TO REQ;
          SUBSCRIBE_3.IND TO REQ;
          SUBSCRIBE_4.IND TO REQ;
          SUBSCRIBE_5.IND TO REQ;
          SUBSCRIBE_6.IND TO REQ;
          SUBSCRIBE_7.IND TO REQ;
          SUBSCRIBE_8.IND TO REQ;
          SUBSCRIBE_9.IND TO REQ;
          SUBSCRIBE_10.IND TO REQ;
          SUBSCRIBE_11.IND TO REQ;
          SUBSCRIBE_12.IND TO REQ;
          SUBSCRIBE_13.IND TO REQ;
          SUBSCRIBE_14.IND TO REQ;
          SUBSCRIBE_15.IND TO REQ;
          SUBSCRIBE_16.IND TO REQ;
          SUBSCRIBE_17.IND TO REQ;
          SUBSCRIBE_18.IND TO REQ;
          SUBSCRIBE_19.IND TO REQ;
          SUBSCRIBE_20.IND TO REQ;
          SUBSCRIBE_21.IND TO REQ;
          SUBSCRIBE_22.IND TO REQ;
          SUBSCRIBE_23.IND TO REQ;
          SUBSCRIBE_24.IND TO REQ;
          SUBSCRIBE_25.IND TO REQ;
          SUBSCRIBE_26.IND TO REQ;
          SUBSCRIBE_27.IND TO REQ;
          SUBSCRIBE_28.IND TO REQ;
          SUBSCRIBE_29.IND TO REQ;
          SUBSCRIBE_30.IND TO REQ;
          SUBSCRIBE_1.INITO TO SUBSCRIBE_2.INIT;
          SUBSCRIBE_2.INITO TO SUBSCRIBE_3.INIT;
          SUBSCRIBE_3.INITO TO SUBSCRIBE_4.INIT;
          SUBSCRIBE_4.INITO TO SUBSCRIBE_5.INIT;
          SUBSCRIBE_5.INITO TO SUBSCRIBE_6.INIT;
          SUBSCRIBE_6.INITO TO SUBSCRIBE_7.INIT;
          SUBSCRIBE_7.INITO TO SUBSCRIBE_8.INIT;
          SUBSCRIBE_8.INITO TO SUBSCRIBE_9.INIT;
          SUBSCRIBE_9.INITO TO SUBSCRIBE_10.INIT;
          SUBSCRIBE_10.INITO TO SUBSCRIBE_11.INIT;
          SUBSCRIBE_11.INITO TO SUBSCRIBE_12.INIT;
          SUBSCRIBE_13.INITO TO SUBSCRIBE_14.INIT;
          SUBSCRIBE_15.INITO TO SUBSCRIBE_16.INIT;
          SUBSCRIBE_16.INITO TO SUBSCRIBE_17.INIT;
          SUBSCRIBE_17.INITO TO SUBSCRIBE_18.INIT;
          SUBSCRIBE_18.INITO TO SUBSCRIBE_19.INIT;
          SUBSCRIBE_19.INITO TO SUBSCRIBE_20.INIT;
          SUBSCRIBE_20.INITO TO SUBSCRIBE_21.INIT;
          SUBSCRIBE_21.INITO TO SUBSCRIBE_22.INIT;
          SUBSCRIBE_22.INITO TO SUBSCRIBE_23.INIT;
          SUBSCRIBE_23.INITO TO SUBSCRIBE_24.INIT;
          SUBSCRIBE_24.INITO TO SUBSCRIBE_25.INIT;
          SUBSCRIBE_25.INITO TO SUBSCRIBE_26.INIT;
          SUBSCRIBE_26.INITO TO SUBSCRIBE_27.INIT;
          SUBSCRIBE_27.INITO TO SUBSCRIBE_28.INIT;
          SUBSCRIBE_28.INITO TO SUBSCRIBE_29.INIT;
          SUBSCRIBE_29.INITO TO SUBSCRIBE_30.INIT;
          INIT TO SUBSCRIBE_1.INIT;
          SUBSCRIBE_12.INITO TO SUBSCRIBE_13.INIT;
        END_CONNECTIONS
        DATA_CONNECTIONS
          SUBSCRIBE_30.RD_1 TO BOOL30;
          SUBSCRIBE_29.RD_1 TO BOOL29;
          SUBSCRIBE_28.RD_1 TO BOOL28;
          SUBSCRIBE_27.RD_1 TO BOOL27;
          SUBSCRIBE_26.RD_1 TO BOOL26;
          SUBSCRIBE_25.RD_1 TO BOOL25;
          SUBSCRIBE_24.RD_1 TO BOOL24;
          SUBSCRIBE_23.RD_1 TO BOOL23;
          SUBSCRIBE_22.RD_1 TO BOOL22;
          SUBSCRIBE_21.RD_1 TO BOOL21;
          SUBSCRIBE_20.RD_1 TO BOOL20;
          SUBSCRIBE_19.RD_1 TO BOOL19;
          SUBSCRIBE_18.RD_1 TO BOOL18;
          SUBSCRIBE_17.RD_1 TO BOOL17;
          SUBSCRIBE_16.RD_1 TO BOOL16;
          SUBSCRIBE_15.RD_1 TO BOOL15;
          SUBSCRIBE_14.RD_1 TO BOOL14;
          SUBSCRIBE_13.RD_1 TO BOOL13;
          SUBSCRIBE_12.RD_1 TO BOOL12;
          SUBSCRIBE_11.RD_1 TO BOOL11;
          SUBSCRIBE_10.RD_1 TO BOOL10;
          SUBSCRIBE_9.RD_1 TO BOOL9;
          SUBSCRIBE_8.RD_1 TO BOOL8;
          SUBSCRIBE_7.RD_1 TO BOOL7;
          SUBSCRIBE_6.RD_1 TO BOOL6;
          SUBSCRIBE_5.RD_1 TO BOOL5;
          SUBSCRIBE_1.RD_1 TO WORD1;
          SUBSCRIBE_2.RD_1 TO WORD2;
          SUBSCRIBE_3.RD_1 TO WORD3;
          SUBSCRIBE_4.RD_1 TO WORD4;
        END_CONNECTIONS
      END_SUBAPPLICATION
      EVENT_CONNECTIONS
        INIT TO IOs_Subscriptions.INIT;
        IOs_Subscriptions.REQ TO F_WORD_TO_DINT.REQ;
        IOs_Subscriptions.REQ TO F_WORD_TO_DINT_2.REQ;
        IOs_Subscriptions.REQ TO BOOL2BOOL.REQ;
        IOs_Subscriptions.REQ TO BOOL2BOOL_1.REQ;
        IOs_Subscriptions.REQ TO BOOL2BOOL_2.REQ;
        IOs_Subscriptions.REQ TO BOOL2BOOL_3.REQ;
        IOs_Subscriptions.REQ TO BOOL2BOOL_4.REQ;
        IOs_Subscriptions.REQ TO BOOL2BOOL_5.REQ;
        IOs_Subscriptions.REQ TO BOOL2BOOL_8.REQ;
        IOs_Subscriptions.REQ TO BOOL2BOOL_10.REQ;
        IOs_Subscriptions.REQ TO BOOL2BOOL_11.REQ;
        SUBSCRIBE_7.IND TO BOOL2BOOL_14.REQ;
        SUBSCRIBE_7.IND TO BOOL2BOOL_15.REQ;
        SUBSCRIBE_7.IND TO BOOL2BOOL_16.REQ;
        SUBSCRIBE_7.IND TO BOOL2BOOL_17.REQ;
        SUBSCRIBE_7.IND TO BOOL2BOOL_18.REQ;
        PUBLISH_1.INITO TO PUBLISH_2.INIT;
        PUBLISH_2.INITO TO PUBLISH_3.INIT;
        PUBLISH_3.INITO TO PUBLISH_4.INIT;
        PUBLISH_4.INITO TO PUBLISH_5.INIT;
        PUBLISH_5.INITO TO PUBLISH_6.INIT;
        BOOL2BOOL_14.CNF TO PUBLISH_3.REQ;
        BOOL2BOOL_15.CNF TO PUBLISH_4.REQ;
        BOOL2BOOL_16.CNF TO PUBLISH_5.REQ;
        BOOL2BOOL_17.CNF TO PUBLISH_6.REQ;
        PUBLISH_6.INITO TO PUBLISH_7.INIT;
        BOOL2BOOL_18.CNF TO PUBLISH_7.REQ;
        INIT TO PUBLISH_30.INIT;
        F_WORD_TO_DINT.CNF TO PUBLISH_30.REQ;
        F_WORD_TO_DINT_2.CNF TO PUBLISH_30.REQ;
        BOOL2BOOL.CNF TO PUBLISH_30.REQ;
        BOOL2BOOL_1.CNF TO PUBLISH_30.REQ;
        BOOL2BOOL_2.CNF TO PUBLISH_30.REQ;
        BOOL2BOOL_3.CNF TO PUBLISH_30.REQ;
        BOOL2BOOL_4.CNF TO PUBLISH_30.REQ;
        BOOL2BOOL_5.CNF TO PUBLISH_30.REQ;
        BOOL2BOOL_8.CNF TO PUBLISH_30.REQ;
        BOOL2BOOL_10.CNF TO PUBLISH_30.REQ;
        BOOL2BOOL_11.CNF TO PUBLISH_30.REQ;
        PUBLISH_30.INITO TO SUBSCRIBE_7.INIT;
        PUBLISH_30.INITO TO PUBLISH_1.INIT;
        WORD2WORD_1.CNF TO PUBLISH_2.REQ;
        SUBSCRIBE_7.IND TO WORD2WORD_1.REQ;
        WORD2WORD.CNF TO PUBLISH_1.REQ;
        SUBSCRIBE_7.IND TO WORD2WORD.REQ;
        IOs_Subscriptions.REQ TO WORD2WORD_2.REQ;
        IOs_Subscriptions.REQ TO WORD2WORD_3.REQ;
        IOs_Subscriptions.REQ TO BOOL2BOOL_6.REQ;
        IOs_Subscriptions.REQ TO BOOL2BOOL_7.REQ;
      END_CONNECTIONS
      DATA_CONNECTIONS
        IOs_Subscriptions.WORD1 TO F_WORD_TO_DINT.IN;
        IOs_Subscriptions.WORD3 TO F_WORD_TO_DINT_2.IN;
        IOs_Subscriptions.BOOL5 TO BOOL2BOOL.IN;
        IOs_Subscriptions.BOOL6 TO BOOL2BOOL_1.IN;
        IOs_Subscriptions.BOOL7 TO BOOL2BOOL_2.IN;
        IOs_Subscriptions.BOOL8 TO BOOL2BOOL_3.IN;
        IOs_Subscriptions.BOOL9 TO BOOL2BOOL_4.IN;
        IOs_Subscriptions.BOOL10 TO BOOL2BOOL_5.IN;
        IOs_Subscriptions.BOOL13 TO BOOL2BOOL_8.IN;
        IOs_Subscriptions.BOOL15 TO BOOL2BOOL_10.IN;
        IOs_Subscriptions.BOOL16 TO BOOL2BOOL_11.IN;
        SUBSCRIBE_7.RD_3 TO BOOL2BOOL_14.IN;
        SUBSCRIBE_7.RD_4 TO BOOL2BOOL_15.IN;
        SUBSCRIBE_7.RD_5 TO BOOL2BOOL_16.IN;
        SUBSCRIBE_7.RD_6 TO BOOL2BOOL_17.IN;
        SUBSCRIBE_7.RD_7 TO BOOL2BOOL_18.IN;
        BOOL2BOOL_14.OUT TO PUBLISH_3.SD_1;
        BOOL2BOOL_15.OUT TO PUBLISH_4.SD_1;
        BOOL2BOOL_16.OUT TO PUBLISH_5.SD_1;
        BOOL2BOOL_17.OUT TO PUBLISH_6.SD_1;
        BOOL2BOOL_18.OUT TO PUBLISH_7.SD_1;
        F_WORD_TO_DINT.OUT TO PUBLISH_30.SD_1;
        F_WORD_TO_DINT_2.OUT TO PUBLISH_30.SD_2;
        BOOL2BOOL.OUT TO PUBLISH_30.SD_3;
        BOOL2BOOL_1.OUT TO PUBLISH_30.SD_4;
        BOOL2BOOL_2.OUT TO PUBLISH_30.SD_5;
        BOOL2BOOL_3.OUT TO PUBLISH_30.SD_6;
        BOOL2BOOL_4.OUT TO PUBLISH_30.SD_7;
        BOOL2BOOL_5.OUT TO PUBLISH_30.SD_8;
        BOOL2BOOL_8.OUT TO PUBLISH_30.SD_9;
        BOOL2BOOL_10.OUT TO PUBLISH_30.SD_10;
        BOOL2BOOL_11.OUT TO PUBLISH_30.SD_11;
        WORD2WORD_1.OUT TO PUBLISH_2.SD_1;
        SUBSCRIBE_7.RD_2 TO WORD2WORD_1.IN;
        WORD2WORD.OUT TO PUBLISH_1.SD_1;
        SUBSCRIBE_7.RD_1 TO WORD2WORD.IN;
        IOs_Subscriptions.WORD4 TO WORD2WORD_3.IN;
        IOs_Subscriptions.WORD2 TO WORD2WORD_2.IN;
        IOs_Subscriptions.BOOL11 TO BOOL2BOOL_6.IN;
        IOs_Subscriptions.BOOL12 TO BOOL2BOOL_7.IN;
      END_CONNECTIONS
    END_SUBAPPLICATION
  END_APPLICATION
  APPLICATION VDMA_Station1_HierarchicalControl
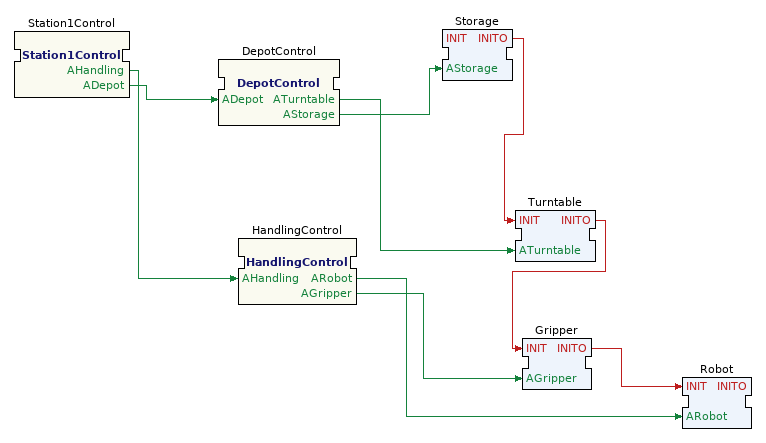
    FBS
      HandlingControl : HandlingControl;
      DepotControl : DepotControl;
      Station1Control : Station1Control;
    END_FBS
    SUBAPPLICATION Robot
      EVENT_INPUT
        INIT;
      END_EVENT
      EVENT_OUTPUT
        INITO;
      END_EVENT
      SOCKETS
        ARobot : ARobot;
      END_SOCKETS
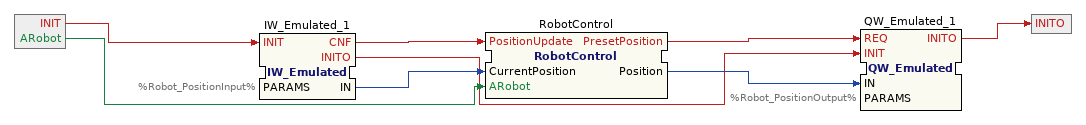
      FBS
        IW_Emulated_1 : IW_Emulated(PARAMS := %Robot_PositionInput%);
        RobotControl : RobotControl;
        QW_Emulated_1 : QW_Emulated(PARAMS := %Robot_PositionOutput%);
      END_FBS
      EVENT_CONNECTIONS
        IW_Emulated_1.CNF TO RobotControl.PositionUpdate;
        RobotControl.PresetPosition TO QW_Emulated_1.REQ;
        IW_Emulated_1.INITO TO QW_Emulated_1.INIT;
        QW_Emulated_1.INITO TO INITO;
        INIT TO IW_Emulated_1.INIT;
      END_CONNECTIONS
      DATA_CONNECTIONS
        IW_Emulated_1.IN TO RobotControl.CurrentPosition;
        RobotControl.Position TO QW_Emulated_1.IN;
      END_CONNECTIONS
      ADAPTER_CONNECTIONS
        ARobot TO RobotControl.ARobot;
      END_CONNECTIONS
    END_SUBAPPLICATION
    SUBAPPLICATION Gripper
      EVENT_INPUT
        INIT;
      END_EVENT
      EVENT_OUTPUT
        INITO;
      END_EVENT
      SOCKETS
        AGripper : AGripper;
      END_SOCKETS
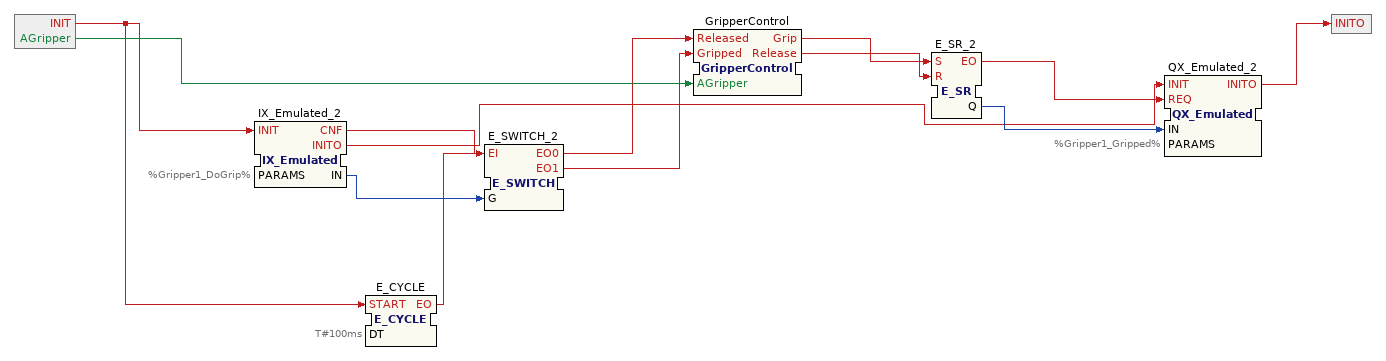
      FBS
        IX_Emulated_2 : IX_Emulated(PARAMS := %Gripper1_DoGrip%);
        E_SWITCH_2 : E_SWITCH;
        GripperControl : GripperControl;
        E_SR_2 : E_SR;
        E_CYCLE : E_CYCLE(DT := T#100ms);
        QX_Emulated_2 : QX_Emulated(PARAMS := %Gripper1_Gripped%);
      END_FBS
      EVENT_CONNECTIONS
        E_SWITCH_2.EO0 TO GripperControl.Released;
        E_SWITCH_2.EO1 TO GripperControl.Gripped;
        GripperControl.Grip TO E_SR_2.S;
        GripperControl.Release TO E_SR_2.R;
        E_CYCLE.EO TO E_SWITCH_2.EI;
        INIT TO E_CYCLE.START;
        IX_Emulated_2.CNF TO E_SWITCH_2.EI;
        INIT TO IX_Emulated_2.INIT;
        IX_Emulated_2.INITO TO QX_Emulated_2.INIT;
        E_SR_2.EO TO QX_Emulated_2.REQ;
        QX_Emulated_2.INITO TO INITO;
      END_CONNECTIONS
      DATA_CONNECTIONS
        IX_Emulated_2.IN TO E_SWITCH_2.G;
        E_SR_2.Q TO QX_Emulated_2.IN;
      END_CONNECTIONS
      ADAPTER_CONNECTIONS
        AGripper TO GripperControl.AGripper;
      END_CONNECTIONS
    END_SUBAPPLICATION
    SUBAPPLICATION Turntable
      EVENT_INPUT
        INIT;
      END_EVENT
      EVENT_OUTPUT
        INITO;
      END_EVENT
      SOCKETS
        ATurntable : ATurntable;
      END_SOCKETS
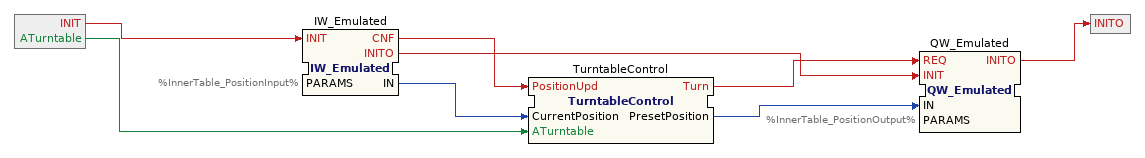
      FBS
        QW_Emulated : QW_Emulated(PARAMS := %InnerTable_PositionOutput%);
        IW_Emulated : IW_Emulated(PARAMS := %InnerTable_PositionInput%);
        TurntableControl : TurntableControl;
      END_FBS
      EVENT_CONNECTIONS
        TurntableControl.Turn TO QW_Emulated.REQ;
        IW_Emulated.CNF TO TurntableControl.PositionUpd;
        IW_Emulated.INITO TO QW_Emulated.INIT;
        INIT TO IW_Emulated.INIT;
        QW_Emulated.INITO TO INITO;
      END_CONNECTIONS
      DATA_CONNECTIONS
        TurntableControl.PresetPosition TO QW_Emulated.IN;
        IW_Emulated.IN TO TurntableControl.CurrentPosition;
      END_CONNECTIONS
      ADAPTER_CONNECTIONS
        ATurntable TO TurntableControl.ATurntable;
      END_CONNECTIONS
    END_SUBAPPLICATION
    SUBAPPLICATION Storage
      EVENT_INPUT
        INIT;
      END_EVENT
      EVENT_OUTPUT
        INITO;
      END_EVENT
      SOCKETS
        AStorage : AStorage;
      END_SOCKETS
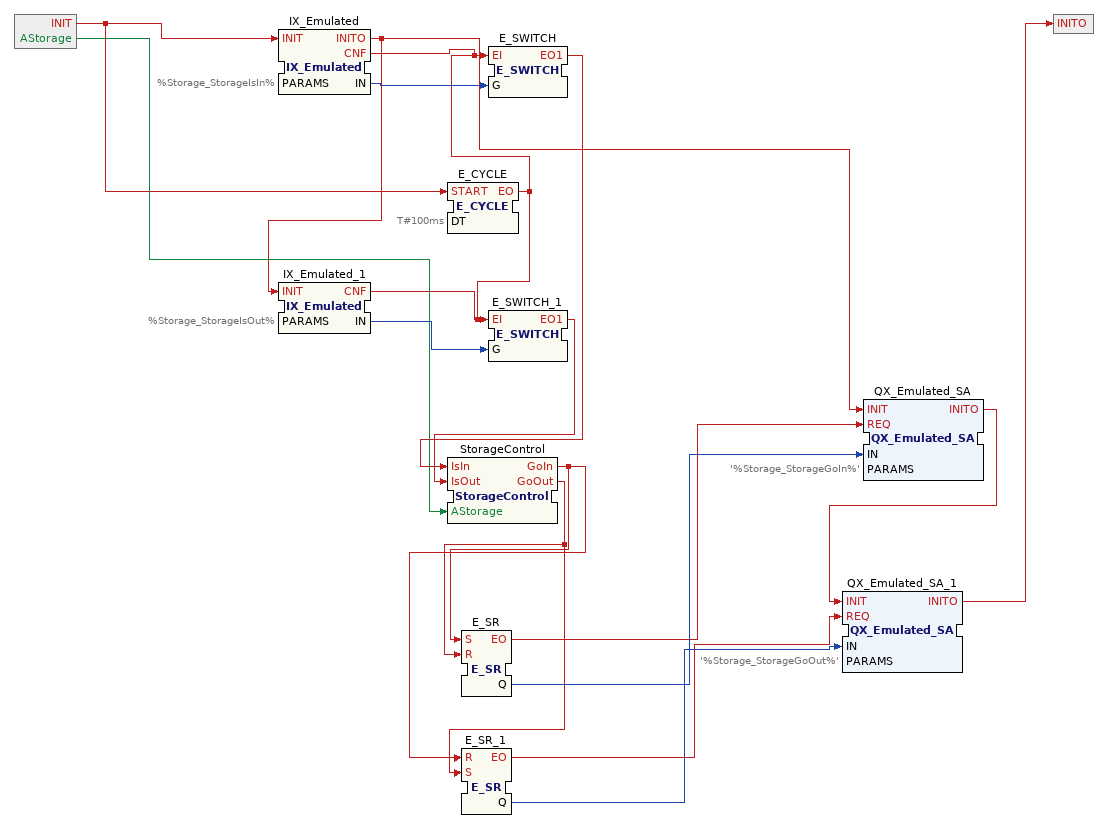
      FBS
        E_SWITCH : E_SWITCH;
        E_SR : E_SR;
        E_SR_1 : E_SR;
        E_SWITCH_1 : E_SWITCH;
        E_CYCLE : E_CYCLE(DT := T#100ms);
        StorageControl : StorageControl;
        IX_Emulated_1 : IX_Emulated(PARAMS := %Storage_StorageIsOut%);
        IX_Emulated : IX_Emulated(PARAMS := %Storage_StorageIsIn%);
      END_FBS
      SUBAPPS
        QX_Emulated_SA : QX_Emulated_SA(PARAMS := '%Storage_StorageGoIn%');
        QX_Emulated_SA_1 : QX_Emulated_SA(PARAMS := '%Storage_StorageGoOut%');
      END_SUBAPPS
      EVENT_CONNECTIONS
        E_CYCLE.EO TO E_SWITCH.EI;
        E_CYCLE.EO TO E_SWITCH_1.EI;
        INIT TO E_CYCLE.START;
        E_SWITCH.EO1 TO StorageControl.IsIn;
        E_SWITCH_1.EO1 TO StorageControl.IsOut;
        StorageControl.GoIn TO E_SR.S;
        StorageControl.GoIn TO E_SR_1.R;
        StorageControl.GoOut TO E_SR.R;
        StorageControl.GoOut TO E_SR_1.S;
        IX_Emulated_1.CNF TO E_SWITCH_1.EI;
        INIT TO IX_Emulated.INIT;
        IX_Emulated.INITO TO IX_Emulated_1.INIT;
        IX_Emulated.CNF TO E_SWITCH.EI;
        IX_Emulated.INITO TO QX_Emulated_SA.INIT;
        E_SR.EO TO QX_Emulated_SA.REQ;
        QX_Emulated_SA.INITO TO QX_Emulated_SA_1.INIT;
        E_SR_1.EO TO QX_Emulated_SA_1.REQ;
        QX_Emulated_SA_1.INITO TO INITO;
      END_CONNECTIONS
      DATA_CONNECTIONS
        IX_Emulated_1.IN TO E_SWITCH_1.G;
        IX_Emulated.IN TO E_SWITCH.G;
        E_SR.Q TO QX_Emulated_SA.IN;
        E_SR_1.Q TO QX_Emulated_SA_1.IN;
      END_CONNECTIONS
      ADAPTER_CONNECTIONS
        AStorage TO StorageControl.AStorage;
      END_CONNECTIONS
    END_SUBAPPLICATION
    EVENT_CONNECTIONS
      Gripper.INITO TO Robot.INIT;
      Turntable.INITO TO Gripper.INIT;
      Storage.INITO TO Turntable.INIT;
    END_CONNECTIONS
    ADAPTER_CONNECTIONS
      HandlingControl.ARobot TO Robot.ARobot;
      HandlingControl.AGripper TO Gripper.AGripper;
      DepotControl.ATurntable TO Turntable.ATurntable;
      DepotControl.AStorage TO Storage.AStorage;
      Station1Control.AHandling TO HandlingControl.AHandling;
      Station1Control.ADepot TO DepotControl.ADepot;
    END_CONNECTIONS
  END_APPLICATION
  APPLICATION VDMA_Station1_SkillbasedControl
